FUNCTION_BLOCK Test_AssertEquals_LINT EXTENDS T_UnitTestBase
VAR
    AssertionUnderTest : T_Assertion;
    LINT_Variable : LINT := 1111;
END_VAR

// Test the assertion...
AssertionUnderTest.AssertEquals_LINT(
    Expected := 2222,
    Actual   := LINT_Variable,
    VariableName := 'LINT_Variable');
 
    
// Assert that the assertion failed...
Assertion.AssertEquals_BOOL(Expected     := TRUE,
                            Actual       := AssertionUnderTest.AssertionFailed,
                            VariableName := 'AssertionUnderTest.AssertionFailed');

// Check the assertion worked...  
CheckAssertion(NextState := 0);

END_FUNCTION_BLOCK

(* stored: Version 1.1.0.1, ProductVersion 3.1.4024.11
   POU Test_AssertEquals_LINT: Id {1485ced9-c1d1-4ec5-b5d9-ba2f49955a42}, SpecialFunc None *)
